// TIA Portal V17 export
// export: Created 2024-12-18T10:10:22.1177395Z, ExportSetting WithDefaults, DisplayName Totally Integrated Automation Portal, DisplayVersion V17, DisplayName TIA Portal Openness, DisplayVersion V17, DisplayName TIA Portal Version Control Interface, DisplayVersion V17, DisplayName STEP 7 Professional, DisplayVersion V17, DisplayName STEP 7 Safety, DisplayVersion V17, DisplayName WinCC Advanced / Unified PC, DisplayVersion V17
FUNCTION_BLOCK "Counter & Pulse"   // FB3, LAD
{ S7_Optimized_Access := 'TRUE' }
VERSION : 0.1
// stored: AutoNumber true, IsIECCheckEnabled false, IsRetainMemResEnabled false, MemoryReserve 100, SetENOAutomatically false, UDAEnableTagReadback false
   VAR_INPUT
      bReset : Bool;
      bChangeHZ : Bool;
      bPuase : Bool;
   END_VAR
   VAR_OUTPUT
      iCvCounter : DInt;
   END_VAR
   VAR
      bCtu : Bool;
      bCtd : Bool;
   END_VAR
   VAR_TEMP   // added for the SCL form of the ladder/FBD networks
      _w1 : Bool;
   END_VAR
BEGIN

REGION Network 1
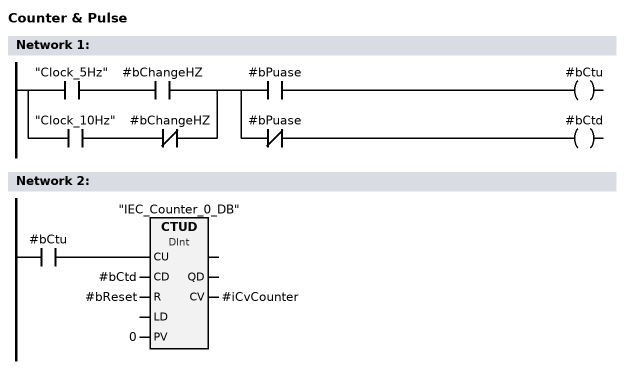
   RUNG wire#powerrail
      Contact( "Clock_5Hz" )
      Contact( #bChangeHZ )
      wire#w1
      Contact( #bPuase )
      Coil( #bCtu )
   END_RUNG
   RUNG wire#powerrail
      Contact( "Clock_10Hz" )
      I_Contact( #bChangeHZ )
   END_RUNG wire#w1
   RUNG wire#w1
      I_Contact( #bPuase )
      Coil( #bCtd )
   END_RUNG
   // the same network as SCL:
   #_w1 := ("Clock_5Hz" AND #bChangeHZ) OR ("Clock_10Hz" AND NOT #bChangeHZ);
   #bCtu := #_w1 AND #bPuase;
   #bCtd := #_w1 AND NOT #bPuase;
END_REGION

REGION Network 2
   RUNG wire#powerrail
      Contact( #bCtu )
      { S7_Templates := "value_type := DInt" } "IEC_Counter_0_DB".CTUD(cd := #bCtd, r := #bReset, ld :=, pv := 0, qd =>, cv => #iCvCounter)
   END_RUNG
   // the same network as SCL:
   "IEC_Counter_0_DB".CTUD(CU := #bCtu, CD := #bCtd, R := #bReset, PV := 0, CV => #iCvCounter);
END_REGION
END_FUNCTION_BLOCK
